// TIA Portal V19 export
FUNCTION "FC900_SafetyIntegration" : Void   // FC900, F_LAD
{ S7_Optimized_Access := 'TRUE' }
// stored: AutoNumber false
BEGIN

REGION Network 1: Bit de reset
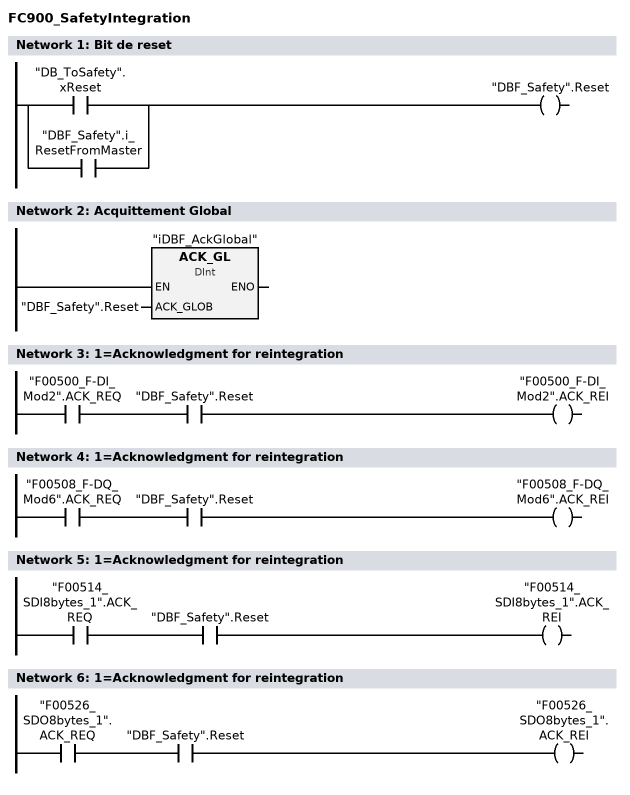
   RUNG wire#powerrail
      Contact( "DB_ToSafety".xReset )
      wire#w1
      Coil( "DBF_Safety".Reset )
   END_RUNG
   RUNG wire#powerrail
      Contact( "DBF_Safety".i_ResetFromMaster )
   END_RUNG wire#w1
   // the same network as SCL:
   "DBF_Safety".Reset := "DB_ToSafety".xReset OR "DBF_Safety".i_ResetFromMaster;
END_REGION

REGION Network 2: Acquittement Global
   RUNG wire#powerrail
      { S7_Templates := "codedbool_type := DInt" } "iDBF_AckGlobal".ACK_GL(ACK_GLOB := "DBF_Safety".Reset)
   END_RUNG
   // the same network as SCL:
   "iDBF_AckGlobal"(ACK_GLOB := "DBF_Safety".Reset);   // ACK_GL
END_REGION

REGION Network 3: 1=Acknowledgment for reintegration
   RUNG wire#powerrail
      Contact( "F00500_F-DI_Mod2".ACK_REQ )
      Contact( "DBF_Safety".Reset )
      Coil( "F00500_F-DI_Mod2".ACK_REI )
   END_RUNG
   // the same network as SCL:
   "F00500_F-DI_Mod2".ACK_REI := "F00500_F-DI_Mod2".ACK_REQ AND "DBF_Safety".Reset;
END_REGION

REGION Network 4: 1=Acknowledgment for reintegration
   RUNG wire#powerrail
      Contact( "F00508_F-DQ_Mod6".ACK_REQ )
      Contact( "DBF_Safety".Reset )
      Coil( "F00508_F-DQ_Mod6".ACK_REI )
   END_RUNG
   // the same network as SCL:
   "F00508_F-DQ_Mod6".ACK_REI := "F00508_F-DQ_Mod6".ACK_REQ AND "DBF_Safety".Reset;
END_REGION

REGION Network 5: 1=Acknowledgment for reintegration
   RUNG wire#powerrail
      Contact( "F00514_SDI8bytes_1".ACK_REQ )
      Contact( "DBF_Safety".Reset )
      Coil( "F00514_SDI8bytes_1".ACK_REI )
   END_RUNG
   // the same network as SCL:
   "F00514_SDI8bytes_1".ACK_REI := "F00514_SDI8bytes_1".ACK_REQ AND "DBF_Safety".Reset;
END_REGION

REGION Network 6: 1=Acknowledgment for reintegration
   RUNG wire#powerrail
      Contact( "F00526_SDO8bytes_1".ACK_REQ )
      Contact( "DBF_Safety".Reset )
      Coil( "F00526_SDO8bytes_1".ACK_REI )
   END_RUNG
   // the same network as SCL:
   "F00526_SDO8bytes_1".ACK_REI := "F00526_SDO8bytes_1".ACK_REQ AND "DBF_Safety".Reset;
END_REGION
END_FUNCTION
